FUNCTION_BLOCK FB_State3 EXTENDS FB_State
VAR_INPUT
END_VAR
VAR_OUTPUT
END_VAR
VAR
END_VAR

END_FUNCTION_BLOCK

(* stored: Version 1.1.0.1, ProductVersion 3.1.4024.12
   POU FB_State3: Id {21520f57-1222-4aa3-8b71-d5f570389035}, SpecialFunc None *)
